ABB RAPID module: P781.mod

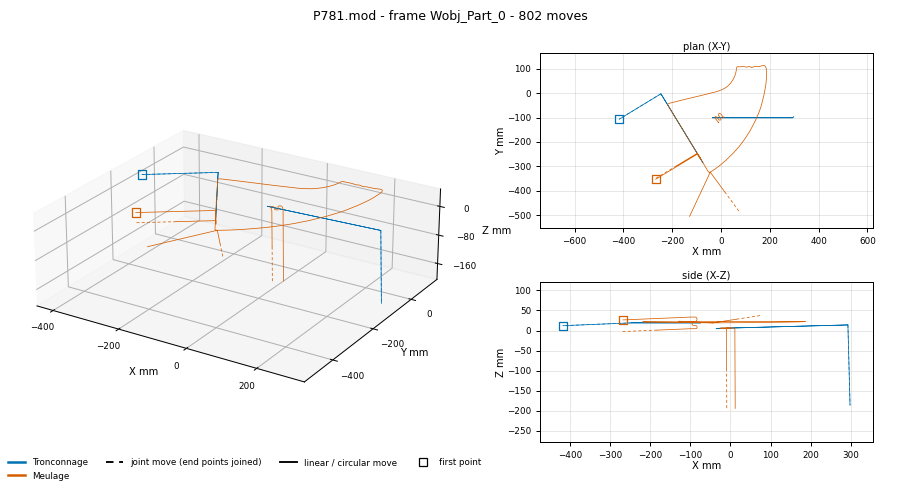
[picture p0: tool path of P781.mod in frame Wobj_Part_0, 802 of 822 moves have a stored position in this frame; points joined in program order, loops and branches not executed]
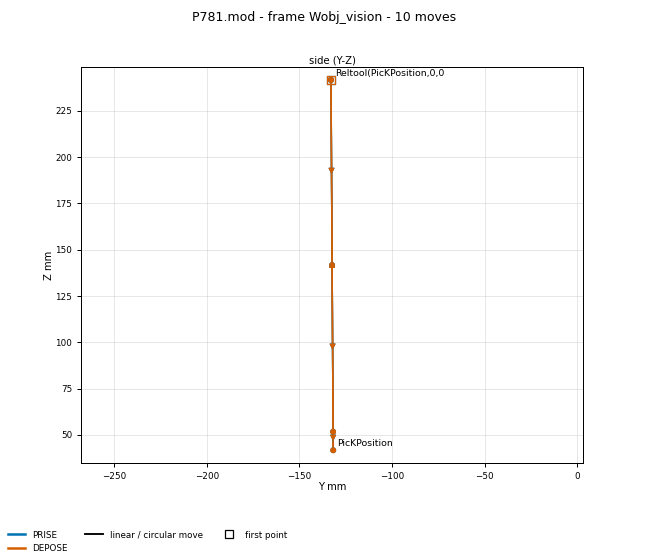
[picture p1: tool path of P781.mod in frame Wobj_vision, 10 of 822 moves have a stored position in this frame; points joined in program order, loops and branches not executed]
MODULE P781

    ! Nom         :P781
    ! Description :
    ! Créé le     :25/05/2023 15:38:47

    LOCAL CONST SPEEDDATA VitesseLente :=[10,500,0,0];
	LOCAL CONST SPEEDDATA VitesseRapide :=[30,500,0,0];
    !
    !Point de prise
    LOCAL PERS Robtarget PicKPosition := [[-23.1582873493958,-131.784324695273,41.7270241668186],[0.00267552588877119,-0.96306839839963,0.269238876085942,0.00159033618135217],[0,0,0,0],[8.999999E+09,8.999999E+09,8.999999E+09,8.999999E+09,8.999999E+09,8.999999E+09]];
	LOCAL PERS Pose Ref := [[0,0,0],[1,0,0,0]];
    !
    !Declaration des points de meulage

    !Tr_meulage_motif_1 : Meulage d'un motif
    LOCAL CONST Robtarget Tr_meulage_motif_1_0 := [[-96.4877265625,-249.765390625,33.67604296875],[0.626544891741501,-0.60457807117296,0.341537876614403,-0.353947359542544],[0,0,0,0],[8.999999E+09,8.999999E+09,8.999999E+09,8.999999E+09,8.999999E+09,8.999999E+09]];
    LOCAL CONST Robtarget Tr_meulage_motif_1_1 := [[-95.966875,-250.619046875,33.676046875],[0.626544891741501,-0.60457807117296,0.341537876614403,-0.353947359542544],[0,0,0,0],[8.999999E+09,8.999999E+09,8.999999E+09,8.999999E+09,8.999999E+09,8.999999E+09]];
    LOCAL CONST Robtarget Tr_meulage_motif_1_2 := [[-95.44603125,-251.4726875,33.6760546875],[0.626544891741501,-0.60457807117296,0.341537876614403,-0.353947359542544],[0,0,0,0],[8.999999E+09,8.999999E+09,8.999999E+09,8.999999E+09,8.999999E+09,8.999999E+09]];
    LOCAL CONST Robtarget Tr_meulage_motif_1_3 := [[-94.9251875,-252.32634375,33.6760625],[0.626544891741501,-0.60457807117296,0.341537876614403,-0.353947359542544],[0,0,0,0],[8.999999E+09,8.999999E+09,8.999999E+09,8.999999E+09,8.999999E+09,8.999999E+09]];
    LOCAL CONST Robtarget Tr_meulage_motif_1_4 := [[-94.40434375,-253.18,33.67606640625],[0.626544891741501,-0.60457807117296,0.341537876614403,-0.353947359542544],[0,0,0,0],[8.999999E+09,8.999999E+09,8.999999E+09,8.999999E+09,8.999999E+09,8.999999E+09]];
    LOCAL CONST Robtarget Tr_meulage_motif_1_5 := [[-93.8834921875,-254.033640625,33.67607421875],[0.626544891741501,-0.60457807117296,0.341537876614403,-0.353947359542544],[0,0,0,0],[8.999999E+09,8.999999E+09,8.999999E+09,8.999999E+09,8.999999E+09,8.999999E+09]];
    LOCAL CONST Robtarget Tr_meulage_motif_1_6 := [[-93.3626484375,-254.887296875,33.676078125],[0.626544891741501,-0.60457807117296,0.341537876614403,-0.353947359542544],[0,0,0,0],[8.999999E+09,8.999999E+09,8.999999E+09,8.999999E+09,8.999999E+09,8.999999E+09]];
    LOCAL CONST Robtarget Tr_meulage_motif_1_7 := [[-92.8418046875,-255.740953125,33.6760859375],[0.626544891741501,-0.60457807117296,0.341537876614403,-0.353947359542544],[0,0,0,0],[8.999999E+09,8.999999E+09,8.999999E+09,8.999999E+09,8.999999E+09,8.999999E+09]];
    LOCAL CONST Robtarget Tr_meulage_motif_1_8 := [[-92.320953125,-256.59459375,33.67608984375],[0.626544891741501,-0.60457807117296,0.341537876614403,-0.353947359542544],[0,0,0,0],[8.999999E+09,8.999999E+09,8.999999E+09,8.999999E+09,8.999999E+09,8.999999E+09]];
    LOCAL CONST Robtarget Tr_meulage_motif_1_9 := [[-91.800109375,-257.44825,33.67609765625],[0.626544891741501,-0.60457807117296,0.341537876614403,-0.353947359542544],[0,0,0,0],[8.999999E+09,8.999999E+09,8.999999E+09,8.999999E+09,8.999999E+09,8.999999E+09]];
    LOCAL CONST Robtarget Tr_meulage_motif_1_10 := [[-91.279265625,-258.30190625,33.6761015625],[0.626544891741501,-0.60457807117296,0.341537876614403,-0.353947359542544],[0,0,0,0],[8.999999E+09,8.999999E+09,8.999999E+09,8.999999E+09,8.999999E+09,8.999999E+09]];
    LOCAL CONST Robtarget Tr_meulage_motif_1_11 := [[-90.758421875,-259.155546875,33.676109375],[0.626544891741501,-0.60457807117296,0.341537876614403,-0.353947359542544],[0,0,0,0],[8.999999E+09,8.999999E+09,8.999999E+09,8.999999E+09,8.999999E+09,8.999999E+09]];
    LOCAL CONST Robtarget Tr_meulage_motif_1_12 := [[-90.2375703125,-260.009203125,33.67611328125],[0.626544891741501,-0.60457807117296,0.341537876614403,-0.353947359542544],[0,0,0,0],[8.999999E+09,8.999999E+09,8.999999E+09,8.999999E+09,8.999999E+09,8.999999E+09]];
    LOCAL CONST Robtarget Tr_meulage_motif_1_13 := [[-89.7167265625,-260.86284375,33.67612109375],[0.626544891741501,-0.60457807117296,0.341537876614403,-0.353947359542544],[0,0,0,0],[8.999999E+09,8.999999E+09,8.999999E+09,8.999999E+09,8.999999E+09,8.999999E+09]];
    LOCAL CONST Robtarget Tr_meulage_motif_1_14 := [[-89.1958828125,-261.7165,33.676125],[0.626544891741501,-0.60457807117296,0.341537876614403,-0.353947359542544],[0,0,0,0],[8.999999E+09,8.999999E+09,8.999999E+09,8.999999E+09,8.999999E+09,8.999999E+09]];
    LOCAL CONST Robtarget Tr_meulage_motif_1_15 := [[-88.67503125,-262.57015625,33.6761328125],[0.626544891741501,-0.60457807117296,0.341537876614403,-0.353947359542544],[0,0,0,0],[8.999999E+09,8.999999E+09,8.999999E+09,8.999999E+09,8.999999E+09,8.999999E+09]];
    LOCAL CONST Robtarget Tr_meulage_motif_1_16 := [[-88.1541875,-263.4238125,33.67613671875],[0.626544891741501,-0.60457807117296,0.341537876614403,-0.353947359542544],[0,0,0,0],[8.999999E+09,8.999999E+09,8.999999E+09,8.999999E+09,8.999999E+09,8.999999E+09]];
    LOCAL CONST Robtarget Tr_meulage_motif_1_17 := [[-87.63334375,-264.27746875,33.67614453125],[0.626544891741501,-0.60457807117296,0.341537876614403,-0.353947359542544],[0,0,0,0],[8.999999E+09,8.999999E+09,8.999999E+09,8.999999E+09,8.999999E+09,8.999999E+09]];
    LOCAL CONST Robtarget Tr_meulage_motif_1_18 := [[-87.1125,-265.13109375,33.6761484375],[0.626544891741501,-0.60457807117296,0.341537876614403,-0.353947359542544],[0,0,0,0],[8.999999E+09,8.999999E+09,8.999999E+09,8.999999E+09,8.999999E+09,8.999999E+09]];
    LOCAL CONST Robtarget Tr_meulage_motif_1_19 := [[-86.59221875,-265.976375,33.56562890625],[0.626544891741501,-0.60457807117296,0.341537876614403,-0.353947359542544],[0,0,0,0],[8.999999E+09,8.999999E+09,8.999999E+09,8.999999E+09,8.999999E+09,8.999999E+09]];
    LOCAL CONST Robtarget Tr_meulage_motif_1_20 := [[-86.0929296875,-266.78053125,33.35457421875],[0.626544891741501,-0.60457807117296,0.341537876614403,-0.353947359542544],[0,0,0,0],[8.999999E+09,8.999999E+09,8.999999E+09,8.999999E+09,8.999999E+09,8.999999E+09]];
    LOCAL CONST Robtarget Tr_meulage_motif_1_21 := [[-85.640671875,-267.5035,33.08290234375],[0.626544891741501,-0.60457807117296,0.341537876614403,-0.353947359542544],[0,0,0,0],[8.999999E+09,8.999999E+09,8.999999E+09,8.999999E+09,8.999999E+09,8.999999E+09]];
    LOCAL CONST Robtarget Tr_meulage_motif_1_22 := [[-85.241828125,-268.13865625,32.807140625],[0.626544891741501,-0.60457807117296,0.341537876614403,-0.353947359542544],[0,0,0,0],[8.999999E+09,8.999999E+09,8.999999E+09,8.999999E+09,8.999999E+09,8.999999E+09]];
    LOCAL CONST Robtarget Tr_meulage_motif_1_23 := [[-84.6499296875,-269.06734375,32.1913984375],[0.626544891741501,-0.60457807117296,0.341537876614403,-0.353947359542544],[0,0,0,0],[8.999999E+09,8.999999E+09,8.999999E+09,8.999999E+09,8.999999E+09,8.999999E+09]];
    LOCAL CONST Robtarget Tr_meulage_motif_1_24 := [[-84.091328125,-269.9259375,31.344267578125],[0.626544891741501,-0.60457807117296,0.341537876614403,-0.353947359542544],[0,0,0,0],[8.999999E+09,8.999999E+09,8.999999E+09,8.999999E+09,8.999999E+09,8.999999E+09]];
    LOCAL CONST Robtarget Tr_meulage_motif_1_25 := [[-83.619234375,-270.630875,30.321025390625],[0.626544891741501,-0.60457807117296,0.341537876614403,-0.353947359542544],[0,0,0,0],[8.999999E+09,8.999999E+09,8.999999E+09,8.999999E+09,8.999999E+09,8.999999E+09]];
    LOCAL CONST Robtarget Tr_meulage_motif_1_26 := [[-83.3316328125,-271.02725,29.2055234375],[0.626544891741501,-0.60457807117296,0.341537876614403,-0.353947359542544],[0,0,0,0],[8.999999E+09,8.999999E+09,8.999999E+09,8.999999E+09,8.999999E+09,8.999999E+09]];
    LOCAL CONST Robtarget Tr_meulage_motif_1_27 := [[-83.2967421875,-271.03765625,28.509982421875],[0.626544891741501,-0.60457807117296,0.341537876614403,-0.353947359542544],[0,0,0,0],[8.999999E+09,8.999999E+09,8.999999E+09,8.999999E+09,8.999999E+09,8.999999E+09]];
    LOCAL CONST Robtarget Tr_meulage_motif_1_28 := [[-83.276984375,-271.025625,27.84913671875],[0.626544891741501,-0.60457807117296,0.341537876614403,-0.353947359542544],[0,0,0,0],[8.999999E+09,8.999999E+09,8.999999E+09,8.999999E+09,8.999999E+09,8.999999E+09]];
    LOCAL CONST Robtarget Tr_meulage_motif_1_29 := [[-83.2858125,-270.96671875,27.188447265625],[0.626544891741501,-0.60457807117296,0.341537876614403,-0.353947359542544],[0,0,0,0],[8.999999E+09,8.999999E+09,8.999999E+09,8.999999E+09,8.999999E+09,8.999999E+09]];
    LOCAL CONST Robtarget Tr_meulage_motif_1_30 := [[-83.512390625,-270.52134375,26.087369140625],[0.626544891741501,-0.60457807117296,0.341537876614403,-0.353947359542544],[0,0,0,0],[8.999999E+09,8.999999E+09,8.999999E+09,8.999999E+09,8.999999E+09,8.999999E+09]];
    LOCAL CONST Robtarget Tr_meulage_motif_1_31 := [[-83.928484375,-269.77175,25.081357421875],[0.626544891741501,-0.60457807117296,0.341537876614403,-0.353947359542544],[0,0,0,0],[8.999999E+09,8.999999E+09,8.999999E+09,8.999999E+09,8.999999E+09,8.999999E+09]];
    LOCAL CONST Robtarget Tr_meulage_motif_1_32 := [[-84.4367578125,-268.883,24.252982421875],[0.626544891741501,-0.60457807117296,0.341537876614403,-0.353947359542544],[0,0,0,0],[8.999999E+09,8.999999E+09,8.999999E+09,8.999999E+09,8.999999E+09,8.999999E+09]];
    LOCAL CONST Robtarget Tr_meulage_motif_1_33 := [[-84.782796875,-268.28925,23.857470703125],[0.626544891741501,-0.60457807117296,0.341537876614403,-0.353947359542544],[0,0,0,0],[8.999999E+09,8.999999E+09,8.999999E+09,8.999999E+09,8.999999E+09,8.999999E+09]];
    LOCAL CONST Robtarget Tr_meulage_motif_1_34 := [[-85.371453125,-267.29171875,23.370232421875],[0.626544891741501,-0.60457807117296,0.341537876614403,-0.353947359542544],[0,0,0,0],[8.999999E+09,8.999999E+09,8.999999E+09,8.999999E+09,8.999999E+09,8.999999E+09]];
    LOCAL CONST Robtarget Tr_meulage_motif_1_35 := [[-85.8036953125,-266.56553125,23.106294921875],[0.626544891741501,-0.60457807117296,0.341537876614403,-0.353947359542544],[0,0,0,0],[8.999999E+09,8.999999E+09,8.999999E+09,8.999999E+09,8.999999E+09,8.999999E+09]];
    LOCAL CONST Robtarget Tr_meulage_motif_1_36 := [[-86.283015625,-265.76621875,22.9019453125],[0.626544891741501,-0.60457807117296,0.341537876614403,-0.353947359542544],[0,0,0,0],[8.999999E+09,8.999999E+09,8.999999E+09,8.999999E+09,8.999999E+09,8.999999E+09]];
    LOCAL CONST Robtarget Tr_meulage_motif_1_37 := [[-86.791015625,-264.9263125,22.7934140625],[0.626544891741501,-0.60457807117296,0.341537876614403,-0.353947359542544],[0,0,0,0],[8.999999E+09,8.999999E+09,8.999999E+09,8.999999E+09,8.999999E+09,8.999999E+09]];
    LOCAL CONST Robtarget Tr_meulage_motif_1_38 := [[-87.3046796875,-264.077,22.682880859375],[0.626544891741501,-0.60457807117296,0.341537876614403,-0.353947359542544],[0,0,0,0],[8.999999E+09,8.999999E+09,8.999999E+09,8.999999E+09,8.999999E+09,8.999999E+09]];
    LOCAL CONST Robtarget Tr_meulage_motif_1_39 := [[-87.8255234375,-263.22334375,22.682875],[0.626544891741501,-0.60457807117296,0.341537876614403,-0.353947359542544],[0,0,0,0],[8.999999E+09,8.999999E+09,8.999999E+09,8.999999E+09,8.999999E+09,8.999999E+09]];
    LOCAL CONST Robtarget Tr_meulage_motif_1_40 := [[-88.346375,-262.3696875,22.682869140625],[0.626544891741501,-0.60457807117296,0.341537876614403,-0.353947359542544],[0,0,0,0],[8.999999E+09,8.999999E+09,8.999999E+09,8.999999E+09,8.999999E+09,8.999999E+09]];
    LOCAL CONST Robtarget Tr_meulage_motif_1_41 := [[-88.86721875,-261.516046875,22.68286328125],[0.626544891741501,-0.60457807117296,0.341537876614403,-0.353947359542544],[0,0,0,0],[8.999999E+09,8.999999E+09,8.999999E+09,8.999999E+09,8.999999E+09,8.999999E+09]];
    LOCAL CONST Robtarget Tr_meulage_motif_1_42 := [[-89.3880625,-260.662390625,22.682857421875],[0.626544891741501,-0.60457807117296,0.341537876614403,-0.353947359542544],[0,0,0,0],[8.999999E+09,8.999999E+09,8.999999E+09,8.999999E+09,8.999999E+09,8.999999E+09]];
    LOCAL CONST Robtarget Tr_meulage_motif_1_43 := [[-89.9089140625,-259.80875,22.6828515625],[0.626544891741501,-0.60457807117296,0.341537876614403,-0.353947359542544],[0,0,0,0],[8.999999E+09,8.999999E+09,8.999999E+09,8.999999E+09,8.999999E+09,8.999999E+09]];
    LOCAL CONST Robtarget Tr_meulage_motif_1_44 := [[-90.4297578125,-258.95509375,22.682845703125],[0.626544891741501,-0.60457807117296,0.341537876614403,-0.353947359542544],[0,0,0,0],[8.999999E+09,8.999999E+09,8.999999E+09,8.999999E+09,8.999999E+09,8.999999E+09]];
    LOCAL CONST Robtarget Tr_meulage_motif_1_45 := [[-90.9506015625,-258.1014375,22.68283984375],[0.626544891741501,-0.60457807117296,0.341537876614403,-0.353947359542544],[0,0,0,0],[8.999999E+09,8.999999E+09,8.999999E+09,8.999999E+09,8.999999E+09,8.999999E+09]];
    LOCAL CONST Robtarget Tr_meulage_motif_1_46 := [[-91.4714453125,-257.247796875,22.682833984375],[0.626544891741501,-0.60457807117296,0.341537876614403,-0.353947359542544],[0,0,0,0],[8.999999E+09,8.999999E+09,8.999999E+09,8.999999E+09,8.999999E+09,8.999999E+09]];
    LOCAL CONST Robtarget Tr_meulage_motif_1_47 := [[-91.992296875,-256.394140625,22.682828125],[0.626544891741501,-0.60457807117296,0.341537876614403,-0.353947359542544],[0,0,0,0],[8.999999E+09,8.999999E+09,8.999999E+09,8.999999E+09,8.999999E+09,8.999999E+09]];
    LOCAL CONST Robtarget Tr_meulage_motif_1_48 := [[-92.513140625,-255.5405,22.682822265625],[0.626544891741501,-0.60457807117296,0.341537876614403,-0.353947359542544],[0,0,0,0],[8.999999E+09,8.999999E+09,8.999999E+09,8.999999E+09,8.999999E+09,8.999999E+09]];
    LOCAL CONST Robtarget Tr_meulage_motif_1_49 := [[-93.0268046875,-254.691171875,22.572291015625],[0.626544891741501,-0.60457807117296,0.341537876614403,-0.353947359542544],[0,0,0,0],[8.999999E+09,8.999999E+09,8.999999E+09,8.999999E+09,8.999999E+09,8.999999E+09]];
    LOCAL CONST Robtarget Tr_meulage_motif_1_50 := [[-93.5134765625,-253.87934375,22.3612265625],[0.626544891741501,-0.60457807117296,0.341537876614403,-0.353947359542544],[0,0,0,0],[8.999999E+09,8.999999E+09,8.999999E+09,8.999999E+09,8.999999E+09,8.999999E+09]];
    LOCAL CONST Robtarget Tr_meulage_motif_1_51 := [[-93.9494921875,-253.14646875,22.089544921875],[0.626544891741501,-0.60457807117296,0.341537876614403,-0.353947359542544],[0,0,0,0],[8.999999E+09,8.999999E+09,8.999999E+09,8.999999E+09,8.999999E+09,8.999999E+09]];
    LOCAL CONST Robtarget Tr_meulage_motif_1_52 := [[-94.310984375,-252.533546875,21.7855703125],[0.626544891741501,-0.60457807117296,0.341537876614403,-0.353947359542544],[0,0,0,0],[8.999999E+09,8.999999E+09,8.999999E+09,8.999999E+09,8.999999E+09,8.999999E+09]];
    LOCAL CONST Robtarget Tr_meulage_motif_1_53 := [[-94.8299921875,-251.63840625,21.123439453125],[0.626544891741501,-0.60457807117296,0.341537876614403,-0.353947359542544],[0,0,0,0],[8.999999E+09,8.999999E+09,8.999999E+09,8.999999E+09,8.999999E+09,8.999999E+09]];
    LOCAL CONST Robtarget Tr_meulage_motif_1_54 := [[-95.2728125,-250.85203125,20.222048828125],[0.626544891741501,-0.60457807117296,0.341537876614403,-0.353947359542544],[0,0,0,0],[8.999999E+09,8.999999E+09,8.999999E+09,8.999999E+09,8.999999E+09,8.999999E+09]];
    LOCAL CONST Robtarget Tr_meulage_motif_1_55 := [[-95.5201953125,-250.376296875,19.176654296875],[0.626544891741501,-0.60457807117296,0.341537876614403,-0.353947359542544],[0,0,0,0],[8.999999E+09,8.999999E+09,8.999999E+09,8.999999E+09,8.999999E+09,8.999999E+09]];
    LOCAL CONST Robtarget Tr_meulage_motif_1_56 := [[-95.5957265625,-250.205921875,18.483859375],[0.626544891741501,-0.60457807117296,0.341537876614403,-0.353947359542544],[0,0,0,0],[8.999999E+09,8.999999E+09,8.999999E+09,8.999999E+09,8.999999E+09,8.999999E+09]];
    LOCAL CONST Robtarget Tr_meulage_motif_1_57 := [[-95.60596875,-250.137390625,17.71433203125],[0.626544891741501,-0.60457807117296,0.341537876614403,-0.353947359542544],[0,0,0,0],[8.999999E+09,8.999999E+09,8.999999E+09,8.999999E+09,8.999999E+09,8.999999E+09]];
    LOCAL CONST Robtarget Tr_meulage_motif_1_58 := [[-95.5481015625,-250.1805,16.944927734375],[0.626544891741501,-0.60457807117296,0.341537876614403,-0.353947359542544],[0,0,0,0],[8.999999E+09,8.999999E+09,8.999999E+09,8.999999E+09,8.999999E+09,8.999999E+09]];
    LOCAL CONST Robtarget Tr_meulage_motif_1_59 := [[-95.2964453125,-250.518484375,15.837359375],[0.626544891741501,-0.60457807117296,0.341537876614403,-0.353947359542544],[0,0,0,0],[8.999999E+09,8.999999E+09,8.999999E+09,8.999999E+09,8.999999E+09,8.999999E+09]];
    LOCAL CONST Robtarget Tr_meulage_motif_1_60 := [[-95.06315625,-250.8615,15.252033203125],[0.626544891741501,-0.60457807117296,0.341537876614403,-0.353947359542544],[0,0,0,0],[8.999999E+09,8.999999E+09,8.999999E+09,8.999999E+09,8.999999E+09,8.999999E+09]];
    LOCAL CONST Robtarget Tr_meulage_motif_1_61 := [[-94.57459375,-251.602625,14.36545703125],[0.626544891741501,-0.60457807117296,0.341537876614403,-0.353947359542544],[0,0,0,0],[8.999999E+09,8.999999E+09,8.999999E+09,8.999999E+09,8.999999E+09,8.999999E+09]];
    LOCAL CONST Robtarget Tr_meulage_motif_1_62 := [[-94.2571640625,-252.095046875,13.95140234375],[0.626544891741501,-0.60457807117296,0.341537876614403,-0.353947359542544],[0,0,0,0],[8.999999E+09,8.999999E+09,8.999999E+09,8.999999E+09,8.999999E+09,8.999999E+09]];
    LOCAL CONST Robtarget Tr_meulage_motif_1_63 := [[-93.6586484375,-253.0394375,13.4076484375],[0.626544891741501,-0.60457807117296,0.341537876614403,-0.353947359542544],[0,0,0,0],[8.999999E+09,8.999999E+09,8.999999E+09,8.999999E+09,8.999999E+09,8.999999E+09]];
    LOCAL CONST Robtarget Tr_meulage_motif_1_64 := [[-93.2198125,-253.7388125,13.112333984375],[0.626544891741501,-0.60457807117296,0.341537876614403,-0.353947359542544],[0,0,0,0],[8.999999E+09,8.999999E+09,8.999999E+09,8.999999E+09,8.999999E+09,8.999999E+09]];
    LOCAL CONST Robtarget Tr_meulage_motif_1_65 := [[-92.7282734375,-254.5306875,12.90799609375],[0.626544891741501,-0.60457807117296,0.341537876614403,-0.353947359542544],[0,0,0,0],[8.999999E+09,8.999999E+09,8.999999E+09,8.999999E+09,8.999999E+09,8.999999E+09]];
    LOCAL CONST Robtarget Tr_meulage_motif_1_66 := [[-92.2137890625,-255.366625,12.799474609375],[0.626544891741501,-0.60457807117296,0.341537876614403,-0.353947359542544],[0,0,0,0],[8.999999E+09,8.999999E+09,8.999999E+09,8.999999E+09,8.999999E+09,8.999999E+09]];
    LOCAL CONST Robtarget Tr_meulage_motif_1_67 := [[-91.6935078125,-256.21190625,12.6889541015625],[0.626544891741501,-0.60457807117296,0.341537876614403,-0.353947359542544],[0,0,0,0],[8.999999E+09,8.999999E+09,8.999999E+09,8.999999E+09,8.999999E+09,8.999999E+09]];
    LOCAL CONST Robtarget Tr_meulage_motif_1_68 := [[-91.1726640625,-257.0655625,12.6889599609375],[0.626544891741501,-0.60457807117296,0.341537876614403,-0.353947359542544],[0,0,0,0],[8.999999E+09,8.999999E+09,8.999999E+09,8.999999E+09,8.999999E+09,8.999999E+09]];
    LOCAL CONST Robtarget Tr_meulage_motif_1_69 := [[-90.6518203125,-257.91921875,12.6889658203125],[0.626544891741501,-0.60457807117296,0.341537876614403,-0.353947359542544],[0,0,0,0],[8.999999E+09,8.999999E+09,8.999999E+09,8.999999E+09,8.999999E+09,8.999999E+09]];
    LOCAL CONST Robtarget Tr_meulage_motif_1_70 := [[-90.1309765625,-258.772859375,12.6889716796875],[0.626544891741501,-0.60457807117296,0.341537876614403,-0.353947359542544],[0,0,0,0],[8.999999E+09,8.999999E+09,8.999999E+09,8.999999E+09,8.999999E+09,8.999999E+09]];
    LOCAL CONST Robtarget Tr_meulage_motif_1_71 := [[-89.610125,-259.626515625,12.6889775390625],[0.626544891741501,-0.60457807117296,0.341537876614403,-0.353947359542544],[0,0,0,0],[8.999999E+09,8.999999E+09,8.999999E+09,8.999999E+09,8.999999E+09,8.999999E+09]];
    LOCAL CONST Robtarget Tr_meulage_motif_1_72 := [[-89.08928125,-260.480171875,12.6889833984375],[0.626544891741501,-0.60457807117296,0.341537876614403,-0.353947359542544],[0,0,0,0],[8.999999E+09,8.999999E+09,8.999999E+09,8.999999E+09,8.999999E+09,8.999999E+09]];
    LOCAL CONST Robtarget Tr_meulage_motif_1_73 := [[-88.5684375,-261.3338125,12.6889892578125],[0.626544891741501,-0.60457807117296,0.341537876614403,-0.353947359542544],[0,0,0,0],[8.999999E+09,8.999999E+09,8.999999E+09,8.999999E+09,8.999999E+09,8.999999E+09]];
    LOCAL CONST Robtarget Tr_meulage_motif_1_74 := [[-88.0475859375,-262.18746875,12.6889951171875],[0.626544891741501,-0.60457807117296,0.341537876614403,-0.353947359542544],[0,0,0,0],[8.999999E+09,8.999999E+09,8.999999E+09,8.999999E+09,8.999999E+09,8.999999E+09]];
    LOCAL CONST Robtarget Tr_meulage_motif_1_75 := [[-87.5267421875,-263.041125,12.6890009765625],[0.626544891741501,-0.60457807117296,0.341537876614403,-0.353947359542544],[0,0,0,0],[8.999999E+09,8.999999E+09,8.999999E+09,8.999999E+09,8.999999E+09,8.999999E+09]];
    LOCAL CONST Robtarget Tr_meulage_motif_1_76 := [[-87.0058984375,-263.89478125,12.6890068359375],[0.626544891741501,-0.60457807117296,0.341537876614403,-0.353947359542544],[0,0,0,0],[8.999999E+09,8.999999E+09,8.999999E+09,8.999999E+09,8.999999E+09,8.999999E+09]];
    LOCAL CONST Robtarget Tr_meulage_motif_1_77 := [[-86.4850546875,-264.74840625,12.6890126953125],[0.626544891741501,-0.60457807117296,0.341537876614403,-0.353947359542544],[0,0,0,0],[8.999999E+09,8.999999E+09,8.999999E+09,8.999999E+09,8.999999E+09,8.999999E+09]];
    LOCAL CONST Robtarget Tr_meulage_motif_1_78 := [[-85.9647734375,-265.59371875,12.5784931640625],[0.626544891741501,-0.60457807117296,0.341537876614403,-0.353947359542544],[0,0,0,0],[8.999999E+09,8.999999E+09,8.999999E+09,8.999999E+09,8.999999E+09,8.999999E+09]];
    LOCAL CONST Robtarget Tr_meulage_motif_1_79 := [[-85.465484375,-266.39784375,12.3674404296875],[0.626544891741501,-0.60457807117296,0.341537876614403,-0.353947359542544],[0,0,0,0],[8.999999E+09,8.999999E+09,8.999999E+09,8.999999E+09,8.999999E+09,8.999999E+09]];
    LOCAL CONST Robtarget Tr_meulage_motif_1_80 := [[-85.0132265625,-267.1208125,12.0957685546875],[0.626544891741501,-0.60457807117296,0.341537876614403,-0.353947359542544],[0,0,0,0],[8.999999E+09,8.999999E+09,8.999999E+09,8.999999E+09,8.999999E+09,8.999999E+09]];
    LOCAL CONST Robtarget Tr_meulage_motif_1_81 := [[-84.6143828125,-267.75596875,11.82000390625],[0.626544891741501,-0.60457807117296,0.341537876614403,-0.353947359542544],[0,0,0,0],[8.999999E+09,8.999999E+09,8.999999E+09,8.999999E+09,8.999999E+09,8.999999E+09]];
    LOCAL CONST Robtarget Tr_meulage_motif_1_82 := [[-84.022484375,-268.68465625,11.2042626953125],[0.626544891741501,-0.60457807117296,0.341537876614403,-0.353947359542544],[0,0,0,0],[8.999999E+09,8.999999E+09,8.999999E+09,8.999999E+09,8.999999E+09,8.999999E+09]];
    LOCAL CONST Robtarget Tr_meulage_motif_1_83 := [[-83.4974765625,-269.4850625,10.31084765625],[0.626544891741501,-0.60457807117296,0.341537876614403,-0.353947359542544],[0,0,0,0],[8.999999E+09,8.999999E+09,8.999999E+09,8.999999E+09,8.999999E+09,8.999999E+09]];
    LOCAL CONST Robtarget Tr_meulage_motif_1_84 := [[-83.147765625,-269.98525,9.2255166015625],[0.626544891741501,-0.60457807117296,0.341537876614403,-0.353947359542544],[0,0,0,0],[8.999999E+09,8.999999E+09,8.999999E+09,8.999999E+09,8.999999E+09,8.999999E+09]];
    LOCAL CONST Robtarget Tr_meulage_motif_1_85 := [[-83.030171875,-270.11184375,8.2417451171875],[0.626544891741501,-0.60457807117296,0.341537876614403,-0.353947359542544],[0,0,0,0],[8.999999E+09,8.999999E+09,8.999999E+09,8.999999E+09,8.999999E+09,8.999999E+09]];
    LOCAL CONST Robtarget Tr_meulage_motif_1_86 := [[-83.09253125,-269.99590625,8.0372138671875],[0.626544891741501,-0.60457807117296,0.341537876614403,-0.353947359542544],[0,0,0,0],[8.999999E+09,8.999999E+09,8.999999E+09,8.999999E+09,8.999999E+09,8.999999E+09]];
    LOCAL CONST Robtarget Tr_meulage_motif_1_87 := [[-83.1350859375,-269.87734375,7.311251953125],[0.626544891741501,-0.60457807117296,0.341537876614403,-0.353947359542544],[0,0,0,0],[8.999999E+09,8.999999E+09,8.999999E+09,8.999999E+09,8.999999E+09,8.999999E+09]];
    LOCAL CONST Robtarget Tr_meulage_motif_1_88 := [[-83.4633515625,-269.276375,6.37491552734375],[0.626544891741501,-0.60457807117296,0.341537876614403,-0.353947359542544],[0,0,0,0],[8.999999E+09,8.999999E+09,8.999999E+09,8.999999E+09,8.999999E+09,8.999999E+09]];
    LOCAL CONST Robtarget Tr_meulage_motif_1_89 := [[-83.7399296875,-268.79190625,5.9113837890625],[0.626544891741501,-0.60457807117296,0.341537876614403,-0.353947359542544],[0,0,0,0],[8.999999E+09,8.999999E+09,8.999999E+09,8.999999E+09,8.999999E+09,8.999999E+09]];
    LOCAL CONST Robtarget Tr_meulage_motif_1_90 := [[-84.312796875,-267.81734375,5.3812646484375],[0.626544891741501,-0.60457807117296,0.341537876614403,-0.353947359542544],[0,0,0,0],[8.999999E+09,8.999999E+09,8.999999E+09,8.999999E+09,8.999999E+09,8.999999E+09]];
    LOCAL CONST Robtarget Tr_meulage_motif_1_91 := [[-84.7450390625,-267.09115625,5.11732763671875],[0.626544891741501,-0.60457807117296,0.341537876614403,-0.353947359542544],[0,0,0,0],[8.999999E+09,8.999999E+09,8.999999E+09,8.999999E+09,8.999999E+09,8.999999E+09]];
    LOCAL CONST Robtarget Tr_meulage_motif_1_92 := [[-85.224359375,-266.29184375,4.912978515625],[0.626544891741501,-0.60457807117296,0.341537876614403,-0.353947359542544],[0,0,0,0],[8.999999E+09,8.999999E+09,8.999999E+09,8.999999E+09,8.999999E+09,8.999999E+09]];
    LOCAL CONST Robtarget Tr_meulage_motif_1_93 := [[-85.732359375,-265.4519375,4.80444580078125],[0.626544891741501,-0.60457807117296,0.341537876614403,-0.353947359542544],[0,0,0,0],[8.999999E+09,8.999999E+09,8.999999E+09,8.999999E+09,8.999999E+09,8.999999E+09]];
    LOCAL CONST Robtarget Tr_meulage_motif_1_94 := [[-86.2460234375,-264.602625,4.6939140625],[0.626544891741501,-0.60457807117296,0.341537876614403,-0.353947359542544],[0,0,0,0],[8.999999E+09,8.999999E+09,8.999999E+09,8.999999E+09,8.999999E+09,8.999999E+09]];
    LOCAL CONST Robtarget Tr_meulage_motif_1_95 := [[-86.7668671875,-263.749,4.69390771484375],[0.626544891741501,-0.60457807117296,0.341537876614403,-0.353947359542544],[0,0,0,0],[8.999999E+09,8.999999E+09,8.999999E+09,8.999999E+09,8.999999E+09,8.999999E+09]];
    LOCAL CONST Robtarget Tr_meulage_motif_1_96 := [[-87.28771875,-262.89534375,4.69390185546875],[0.626544891741501,-0.60457807117296,0.341537876614403,-0.353947359542544],[0,0,0,0],[8.999999E+09,8.999999E+09,8.999999E+09,8.999999E+09,8.999999E+09,8.999999E+09]];
    LOCAL CONST Robtarget Tr_meulage_motif_1_97 := [[-87.8085625,-262.0416875,4.69389599609375],[0.626544891741501,-0.60457807117296,0.341537876614403,-0.353947359542544],[0,0,0,0],[8.999999E+09,8.999999E+09,8.999999E+09,8.999999E+09,8.999999E+09,8.999999E+09]];
    LOCAL CONST Robtarget Tr_meulage_motif_1_98 := [[-88.32940625,-261.18803125,4.69389013671875],[0.626544891741501,-0.60457807117296,0.341537876614403,-0.353947359542544],[0,0,0,0],[8.999999E+09,8.999999E+09,8.999999E+09,8.999999E+09,8.999999E+09,8.999999E+09]];
    LOCAL CONST Robtarget Tr_meulage_motif_1_99 := [[-88.8502578125,-260.334375,4.69388427734375],[0.626544891741501,-0.60457807117296,0.341537876614403,-0.353947359542544],[0,0,0,0],[8.999999E+09,8.999999E+09,8.999999E+09,8.999999E+09,8.999999E+09,8.999999E+09]];
    LOCAL CONST Robtarget Tr_meulage_motif_1_100 := [[-89.3711015625,-259.480734375,4.69387841796875],[0.626544891741501,-0.60457807117296,0.341537876614403,-0.353947359542544],[0,0,0,0],[8.999999E+09,8.999999E+09,8.999999E+09,8.999999E+09,8.999999E+09,8.999999E+09]];
    LOCAL CONST Robtarget Tr_meulage_motif_1_101 := [[-89.8919453125,-258.627078125,4.69387255859375],[0.626544891741501,-0.60457807117296,0.341537876614403,-0.353947359542544],[0,0,0,0],[8.999999E+09,8.999999E+09,8.999999E+09,8.999999E+09,8.999999E+09,8.999999E+09]];
    LOCAL CONST Robtarget Tr_meulage_motif_1_102 := [[-90.4127890625,-257.7734375,4.69386669921875],[0.626544891741501,-0.60457807117296,0.341537876614403,-0.353947359542544],[0,0,0,0],[8.999999E+09,8.999999E+09,8.999999E+09,8.999999E+09,8.999999E+09,8.999999E+09]];
    LOCAL CONST Robtarget Tr_meulage_motif_1_103 := [[-90.933640625,-256.91978125,4.69386083984375],[0.626544891741501,-0.60457807117296,0.341537876614403,-0.353947359542544],[0,0,0,0],[8.999999E+09,8.999999E+09,8.999999E+09,8.999999E+09,8.999999E+09,8.999999E+09]];
    LOCAL CONST Robtarget Tr_meulage_motif_1_104 := [[-91.454484375,-256.066125,4.69385498046875],[0.626544891741501,-0.60457807117296,0.341537876614403,-0.353947359542544],[0,0,0,0],[8.999999E+09,8.999999E+09,8.999999E+09,8.999999E+09,8.999999E+09,8.999999E+09]];
    LOCAL CONST Robtarget Tr_meulage_motif_1_105 := [[-91.975328125,-255.212484375,4.69384912109375],[0.626544891741501,-0.60457807117296,0.341537876614403,-0.353947359542544],[0,0,0,0],[8.999999E+09,8.999999E+09,8.999999E+09,8.999999E+09,8.999999E+09,8.999999E+09]];
    LOCAL CONST Robtarget Tr_meulage_motif_1_106 := [[-92.4961796875,-254.358828125,4.69384326171875],[0.626544891741501,-0.60457807117296,0.341537876614403,-0.353947359542544],[0,0,0,0],[8.999999E+09,8.999999E+09,8.999999E+09,8.999999E+09,8.999999E+09,8.999999E+09]];
    LOCAL CONST Robtarget Tr_meulage_motif_1_107 := [[-93.0170234375,-253.505171875,4.69383740234375],[0.626544891741501,-0.60457807117296,0.341537876614403,-0.353947359542544],[0,0,0,0],[8.999999E+09,8.999999E+09,8.999999E+09,8.999999E+09,8.999999E+09,8.999999E+09]];
    LOCAL CONST Robtarget Tr_meulage_motif_1_108 := [[-93.5378671875,-252.65153125,4.69383154296875],[0.626544891741501,-0.60457807117296,0.341537876614403,-0.353947359542544],[0,0,0,0],[8.999999E+09,8.999999E+09,8.999999E+09,8.999999E+09,8.999999E+09,8.999999E+09]];
    LOCAL CONST Robtarget Tr_meulage_motif_1_109 := [[-94.0587109375,-251.797875,4.69382568359375],[0.626544891741501,-0.60457807117296,0.341537876614403,-0.353947359542544],[0,0,0,0],[8.999999E+09,8.999999E+09,8.999999E+09,8.999999E+09,8.999999E+09,8.999999E+09]];
    LOCAL CONST Robtarget Tr_meulage_motif_1_110 := [[-94.5795625,-250.94421875,4.69381982421875],[0.626544891741501,-0.60457807117296,0.341537876614403,-0.353947359542544],[0,0,0,0],[8.999999E+09,8.999999E+09,8.999999E+09,8.999999E+09,8.999999E+09,8.999999E+09]];
    LOCAL CONST Robtarget Tr_meulage_motif_1_111 := [[-95.10040625,-250.090578125,4.69381396484375],[0.626544891741501,-0.60457807117296,0.341537876614403,-0.353947359542544],[0,0,0,0],[8.999999E+09,8.999999E+09,8.999999E+09,8.999999E+09,8.999999E+09,8.999999E+09]];
    LOCAL CONST Robtarget Tr_meulage_motif_1_112 := [[-95.62125,-249.236921875,4.69380810546875],[0.626544891741501,-0.60457807117296,0.341537876614403,-0.353947359542544],[0,0,0,0],[8.999999E+09,8.999999E+09,8.999999E+09,8.999999E+09,8.999999E+09,8.999999E+09]];
    LOCAL CONST Robtarget Tr_meulage_motif_1_113 := [[-96.1421015625,-248.383265625,4.6938017578125],[0.626544891741501,-0.60457807117296,0.341537876614403,-0.353947359542544],[0,0,0,0],[8.999999E+09,8.999999E+09,8.999999E+09,8.999999E+09,8.999999E+09,8.999999E+09]];
    LOCAL CONST Robtarget Tr_meulage_motif_1_114 := [[-96.6629453125,-247.529625,4.6937958984375],[0.626544891741501,-0.60457807117296,0.341537876614403,-0.353947359542544],[0,0,0,0],[8.999999E+09,8.999999E+09,8.999999E+09,8.999999E+09,8.999999E+09,8.999999E+09]];
    LOCAL CONST Robtarget Tr_meulage_motif_1_115 := [[-97.1837890625,-246.67596875,4.6937900390625],[0.626544891741501,-0.60457807117296,0.341537876614403,-0.353947359542544],[0,0,0,0],[8.999999E+09,8.999999E+09,8.999999E+09,8.999999E+09,8.999999E+09,8.999999E+09]];

    !Tr_meulage_motif_2 : Meulage d'un motif
    LOCAL CONST Robtarget Tr_meulage_motif_2_0 := [[11.059822265625,-100.7916484375,6.14594775390625],[1.9380529697738E-05,0.00227567224534522,0.00851606674262758,-0.999961148018993],[0,0,0,0],[8.999999E+09,8.999999E+09,8.999999E+09,8.999999E+09,8.999999E+09,8.999999E+09]];
    LOCAL CONST Robtarget Tr_meulage_motif_2_1 := [[10.444326171875,-100.0036640625,6.16165283203125],[1.9380529697738E-05,0.00227567224534522,0.00851606674262758,-0.999961148018993],[0,0,0,0],[8.999999E+09,8.999999E+09,8.999999E+09,8.999999E+09,8.999999E+09,8.999999E+09]];
    LOCAL CONST Robtarget Tr_meulage_motif_2_2 := [[9.828830078125,-99.2156875,6.17735791015625],[1.9380529697738E-05,0.00227567224534522,0.00851606674262758,-0.999961148018993],[0,0,0,0],[8.999999E+09,8.999999E+09,8.999999E+09,8.999999E+09,8.999999E+09,8.999999E+09]];
    LOCAL CONST Robtarget Tr_meulage_motif_2_3 := [[9.2133349609375,-98.427703125,6.19306298828125],[1.9380529697738E-05,0.00227567224534522,0.00851606674262758,-0.999961148018993],[0,0,0,0],[8.999999E+09,8.999999E+09,8.999999E+09,8.999999E+09,8.999999E+09,8.999999E+09]];
    LOCAL CONST Robtarget Tr_meulage_motif_2_4 := [[8.5978388671875,-97.63971875,6.20876806640625],[1.9380529697738E-05,0.00227567224534522,0.00851606674262758,-0.999961148018993],[0,0,0,0],[8.999999E+09,8.999999E+09,8.999999E+09,8.999999E+09,8.999999E+09,8.999999E+09]];
    LOCAL CONST Robtarget Tr_meulage_motif_2_5 := [[7.9823427734375,-96.851734375,6.22447314453125],[1.9380529697738E-05,0.00227567224534522,0.00851606674262758,-0.999961148018993],[0,0,0,0],[8.999999E+09,8.999999E+09,8.999999E+09,8.999999E+09,8.999999E+09,8.999999E+09]];
    LOCAL CONST Robtarget Tr_meulage_motif_2_6 := [[7.3668466796875,-96.06375,6.24017822265625],[1.9380529697738E-05,0.00227567224534522,0.00851606674262758,-0.999961148018993],[0,0,0,0],[8.999999E+09,8.999999E+09,8.999999E+09,8.999999E+09,8.999999E+09,8.999999E+09]];
    LOCAL CONST Robtarget Tr_meulage_motif_2_7 := [[6.75135107421875,-95.275765625,6.2558828125],[1.9380529697738E-05,0.00227567224534522,0.00851606674262758,-0.999961148018993],[0,0,0,0],[8.999999E+09,8.999999E+09,8.999999E+09,8.999999E+09,8.999999E+09,8.999999E+09]];
    LOCAL CONST Robtarget Tr_meulage_motif_2_8 := [[6.13585498046875,-94.48778125,6.271587890625],[1.9380529697738E-05,0.00227567224534522,0.00851606674262758,-0.999961148018993],[0,0,0,0],[8.999999E+09,8.999999E+09,8.999999E+09,8.999999E+09,8.999999E+09,8.999999E+09]];
    LOCAL CONST Robtarget Tr_meulage_motif_2_9 := [[5.520359375,-93.699796875,6.28729296875],[1.9380529697738E-05,0.00227567224534522,0.00851606674262758,-0.999961148018993],[0,0,0,0],[8.999999E+09,8.999999E+09,8.999999E+09,8.999999E+09,8.999999E+09,8.999999E+09]];
    LOCAL CONST Robtarget Tr_meulage_motif_2_10 := [[4.90486328125,-92.9118125,6.302998046875],[1.9380529697738E-05,0.00227567224534522,0.00851606674262758,-0.999961148018993],[0,0,0,0],[8.999999E+09,8.999999E+09,8.999999E+09,8.999999E+09,8.999999E+09,8.999999E+09]];
    LOCAL CONST Robtarget Tr_meulage_motif_2_11 := [[4.28936767578125,-92.123828125,6.318703125],[1.9380529697738E-05,0.00227567224534522,0.00851606674262758,-0.999961148018993],[0,0,0,0],[8.999999E+09,8.999999E+09,8.999999E+09,8.999999E+09,8.999999E+09,8.999999E+09]];
    LOCAL CONST Robtarget Tr_meulage_motif_2_12 := [[3.67387158203125,-91.3358515625,6.334408203125],[1.9380529697738E-05,0.00227567224534522,0.00851606674262758,-0.999961148018993],[0,0,0,0],[8.999999E+09,8.999999E+09,8.999999E+09,8.999999E+09,8.999999E+09,8.999999E+09]];
    LOCAL CONST Robtarget Tr_meulage_motif_2_13 := [[3.05837573242187,-90.5478671875,6.35011279296875],[1.9380529697738E-05,0.00227567224534522,0.00851606674262758,-0.999961148018993],[0,0,0,0],[8.999999E+09,8.999999E+09,8.999999E+09,8.999999E+09,8.999999E+09,8.999999E+09]];
    LOCAL CONST Robtarget Tr_meulage_motif_2_14 := [[2.4428798828125,-89.7598828125,6.36581787109375],[1.9380529697738E-05,0.00227567224534522,0.00851606674262758,-0.999961148018993],[0,0,0,0],[8.999999E+09,8.999999E+09,8.999999E+09,8.999999E+09,8.999999E+09,8.999999E+09]];
    LOCAL CONST Robtarget Tr_meulage_motif_2_15 := [[1.82738403320313,-88.9718984375,6.38152294921875],[1.9380529697738E-05,0.00227567224534522,0.00851606674262758,-0.999961148018993],[0,0,0,0],[8.999999E+09,8.999999E+09,8.999999E+09,8.999999E+09,8.999999E+09,8.999999E+09]];
    LOCAL CONST Robtarget Tr_meulage_motif_2_16 := [[1.21188806152344,-88.1839140625,6.39722802734375],[1.9380529697738E-05,0.00227567224534522,0.00851606674262758,-0.999961148018993],[0,0,0,0],[8.999999E+09,8.999999E+09,8.999999E+09,8.999999E+09,8.999999E+09,8.999999E+09]];
    LOCAL CONST Robtarget Tr_meulage_motif_2_17 := [[0.596392211914063,-87.3959296875,6.41293310546875],[1.9380529697738E-05,0.00227567224534522,0.00851606674262758,-0.999961148018993],[0,0,0,0],[8.999999E+09,8.999999E+09,8.999999E+09,8.999999E+09,8.999999E+09,8.999999E+09]];
    LOCAL CONST Robtarget Tr_meulage_motif_2_18 := [[-0.0191036529541016,-86.6079453125,6.42863818359375],[1.9380529697738E-05,0.00227567224534522,0.00851606674262758,-0.999961148018993],[0,0,0,0],[8.999999E+09,8.999999E+09,8.999999E+09,8.999999E+09,8.999999E+09,8.999999E+09]];
    LOCAL CONST Robtarget Tr_meulage_motif_2_19 := [[-0.717185119628906,-85.893875,6.44274560546875],[1.9380529697738E-05,0.00227567224534522,0.00851606674262758,-0.999961148018993],[0,0,0,0],[8.999999E+09,8.999999E+09,8.999999E+09,8.999999E+09,8.999999E+09,8.999999E+09]];
    LOCAL CONST Robtarget Tr_meulage_motif_2_20 := [[-1.46619714355469,-85.2780078125,6.454783203125],[1.9380529697738E-05,0.00227567224534522,0.00851606674262758,-0.999961148018993],[0,0,0,0],[8.999999E+09,8.999999E+09,8.999999E+09,8.999999E+09,8.999999E+09,8.999999E+09]];
    LOCAL CONST Robtarget Tr_meulage_motif_2_21 := [[-2.20529296875,-84.773359375,6.4645361328125],[1.9380529697738E-05,0.00227567224534522,0.00851606674262758,-0.999961148018993],[0,0,0,0],[8.999999E+09,8.999999E+09,8.999999E+09,8.999999E+09,8.999999E+09,8.999999E+09]];
    LOCAL CONST Robtarget Tr_meulage_motif_2_22 := [[-2.884353515625,-84.35221875,6.47261962890625],[1.9380529697738E-05,0.00227567224534522,0.00851606674262758,-0.999961148018993],[0,0,0,0],[8.999999E+09,8.999999E+09,8.999999E+09,8.999999E+09,8.999999E+09,8.999999E+09]];
    LOCAL CONST Robtarget Tr_meulage_motif_2_23 := [[-4.0476455078125,-83.8637265625,6.48166357421875],[1.9380529697738E-05,0.00227567224534522,0.00851606674262758,-0.999961148018993],[0,0,0,0],[8.999999E+09,8.999999E+09,8.999999E+09,8.999999E+09,8.999999E+09,8.999999E+09]];
    LOCAL CONST Robtarget Tr_meulage_motif_2_24 := [[-5.34590771484375,-83.5785390625,6.4863955078125],[1.9380529697738E-05,0.00227567224534522,0.00851606674262758,-0.999961148018993],[0,0,0,0],[8.999999E+09,8.999999E+09,8.999999E+09,8.999999E+09,8.999999E+09,8.999999E+09]];
    LOCAL CONST Robtarget Tr_meulage_motif_2_25 := [[-6.67459326171875,-83.540640625,6.4860009765625],[1.9380529697738E-05,0.00227567224534522,0.00851606674262758,-0.999961148018993],[0,0,0,0],[8.999999E+09,8.999999E+09,8.999999E+09,8.999999E+09,8.999999E+09,8.999999E+09]];
    LOCAL CONST Robtarget Tr_meulage_motif_2_26 := [[-7.85476318359375,-83.842828125,6.478724609375],[1.9380529697738E-05,0.00227567224534522,0.00851606674262758,-0.999961148018993],[0,0,0,0],[8.999999E+09,8.999999E+09,8.999999E+09,8.999999E+09,8.999999E+09,8.999999E+09]];
    LOCAL CONST Robtarget Tr_meulage_motif_2_27 := [[-8.4199404296875,-84.2497734375,6.46983251953125],[1.9380529697738E-05,0.00227567224534522,0.00851606674262758,-0.999961148018993],[0,0,0,0],[8.999999E+09,8.999999E+09,8.999999E+09,8.999999E+09,8.999999E+09,8.999999E+09]];
    LOCAL CONST Robtarget Tr_meulage_motif_2_28 := [[-8.94109765625,-84.656671875,6.46097998046875],[1.9380529697738E-05,0.00227567224534522,0.00851606674262758,-0.999961148018993],[0,0,0,0],[8.999999E+09,8.999999E+09,8.999999E+09,8.999999E+09,8.999999E+09,8.999999E+09]];
    LOCAL CONST Robtarget Tr_meulage_motif_2_29 := [[-9.4283564453125,-85.10671875,6.45126806640625],[1.9380529697738E-05,0.00227567224534522,0.00851606674262758,-0.999961148018993],[0,0,0,0],[8.999999E+09,8.999999E+09,8.999999E+09,8.999999E+09,8.999999E+09,8.999999E+09]];
    LOCAL CONST Robtarget Tr_meulage_motif_2_30 := [[-9.9900380859375,-86.177265625,6.42869384765625],[1.9380529697738E-05,0.00227567224534522,0.00851606674262758,-0.999961148018993],[0,0,0,0],[8.999999E+09,8.999999E+09,8.999999E+09,8.999999E+09,8.999999E+09,8.999999E+09]];
    LOCAL CONST Robtarget Tr_meulage_motif_2_31 := [[-10.2561494140625,-87.471703125,6.4017646484375],[1.9380529697738E-05,0.00227567224534522,0.00851606674262758,-0.999961148018993],[0,0,0,0],[8.999999E+09,8.999999E+09,8.999999E+09,8.999999E+09,8.999999E+09,8.999999E+09]];
    LOCAL CONST Robtarget Tr_meulage_motif_2_32 := [[-10.2795166015625,-88.7881796875,6.374595703125],[1.9380529697738E-05,0.00227567224534522,0.00851606674262758,-0.999961148018993],[0,0,0,0],[8.999999E+09,8.999999E+09,8.999999E+09,8.999999E+09,8.999999E+09,8.999999E+09]];
    LOCAL CONST Robtarget Tr_meulage_motif_2_33 := [[-10.16851953125,-89.573125,6.3585068359375],[1.9380529697738E-05,0.00227567224534522,0.00851606674262758,-0.999961148018993],[0,0,0,0],[8.999999E+09,8.999999E+09,8.999999E+09,8.999999E+09,8.999999E+09,8.999999E+09]];
    LOCAL CONST Robtarget Tr_meulage_motif_2_34 := [[-9.839921875,-90.785734375,6.333791015625],[1.9380529697738E-05,0.00227567224534522,0.00851606674262758,-0.999961148018993],[0,0,0,0],[8.999999E+09,8.999999E+09,8.999999E+09,8.999999E+09,8.999999E+09,8.999999E+09]];
    LOCAL CONST Robtarget Tr_meulage_motif_2_35 := [[-9.527951171875,-91.6141171875,6.316984375],[1.9380529697738E-05,0.00227567224534522,0.00851606674262758,-0.999961148018993],[0,0,0,0],[8.999999E+09,8.999999E+09,8.999999E+09,8.999999E+09,8.999999E+09,8.999999E+09]];
    LOCAL CONST Robtarget Tr_meulage_motif_2_36 := [[-9.115458984375,-92.4743359375,6.29960986328125],[1.9380529697738E-05,0.00227567224534522,0.00851606674262758,-0.999961148018993],[0,0,0,0],[8.999999E+09,8.999999E+09,8.999999E+09,8.999999E+09,8.999999E+09,8.999999E+09]];
    LOCAL CONST Robtarget Tr_meulage_motif_2_37 := [[-8.5968984375,-93.314609375,6.28274072265625],[1.9380529697738E-05,0.00227567224534522,0.00851606674262758,-0.999961148018993],[0,0,0,0],[8.999999E+09,8.999999E+09,8.999999E+09,8.999999E+09,8.999999E+09,8.999999E+09]];
    LOCAL CONST Robtarget Tr_meulage_motif_2_38 := [[-8.0731435546875,-94.1647890625,6.265671875],[1.9380529697738E-05,0.00227567224534522,0.00851606674262758,-0.999961148018993],[0,0,0,0],[8.999999E+09,8.999999E+09,8.999999E+09,8.999999E+09,8.999999E+09,8.999999E+09]];
    LOCAL CONST Robtarget Tr_meulage_motif_2_39 := [[-7.4576474609375,-94.9527734375,6.249966796875],[1.9380529697738E-05,0.00227567224534522,0.00851606674262758,-0.999961148018993],[0,0,0,0],[8.999999E+09,8.999999E+09,8.999999E+09,8.999999E+09,8.999999E+09,8.999999E+09]];
    LOCAL CONST Robtarget Tr_meulage_motif_2_40 := [[-6.84215185546875,-95.7407578125,6.23426220703125],[1.9380529697738E-05,0.00227567224534522,0.00851606674262758,-0.999961148018993],[0,0,0,0],[8.999999E+09,8.999999E+09,8.999999E+09,8.999999E+09,8.999999E+09,8.999999E+09]];
    LOCAL CONST Robtarget Tr_meulage_motif_2_41 := [[-6.22665576171875,-96.5287421875,6.21855712890625],[1.9380529697738E-05,0.00227567224534522,0.00851606674262758,-0.999961148018993],[0,0,0,0],[8.999999E+09,8.999999E+09,8.999999E+09,8.999999E+09,8.999999E+09,8.999999E+09]];
    LOCAL CONST Robtarget Tr_meulage_motif_2_42 := [[-5.61116015625,-97.3167265625,6.20285205078125],[1.9380529697738E-05,0.00227567224534522,0.00851606674262758,-0.999961148018993],[0,0,0,0],[8.999999E+09,8.999999E+09,8.999999E+09,8.999999E+09,8.999999E+09,8.999999E+09]];
    LOCAL CONST Robtarget Tr_meulage_motif_2_43 := [[-4.9956640625,-98.1047109375,6.18714697265625],[1.9380529697738E-05,0.00227567224534522,0.00851606674262758,-0.999961148018993],[0,0,0,0],[8.999999E+09,8.999999E+09,8.999999E+09,8.999999E+09,8.999999E+09,8.999999E+09]];
    LOCAL CONST Robtarget Tr_meulage_motif_2_44 := [[-4.38016796875,-98.8926953125,6.17144189453125],[1.9380529697738E-05,0.00227567224534522,0.00851606674262758,-0.999961148018993],[0,0,0,0],[8.999999E+09,8.999999E+09,8.999999E+09,8.999999E+09,8.999999E+09,8.999999E+09]];
    LOCAL CONST Robtarget Tr_meulage_motif_2_45 := [[-3.76467236328125,-99.680671875,6.15573681640625],[1.9380529697738E-05,0.00227567224534522,0.00851606674262758,-0.999961148018993],[0,0,0,0],[8.999999E+09,8.999999E+09,8.999999E+09,8.999999E+09,8.999999E+09,8.999999E+09]];
    LOCAL CONST Robtarget Tr_meulage_motif_2_46 := [[-3.14917651367188,-100.46865625,6.1400322265625],[1.9380529697738E-05,0.00227567224534522,0.00851606674262758,-0.999961148018993],[0,0,0,0],[8.999999E+09,8.999999E+09,8.999999E+09,8.999999E+09,8.999999E+09,8.999999E+09]];
    LOCAL CONST Robtarget Tr_meulage_motif_2_47 := [[-2.53368041992187,-101.256640625,6.1243271484375],[1.9380529697738E-05,0.00227567224534522,0.00851606674262758,-0.999961148018993],[0,0,0,0],[8.999999E+09,8.999999E+09,8.999999E+09,8.999999E+09,8.999999E+09,8.999999E+09]];
    LOCAL CONST Robtarget Tr_meulage_motif_2_48 := [[-1.91818469238281,-102.044625,6.1086220703125],[1.9380529697738E-05,0.00227567224534522,0.00851606674262758,-0.999961148018993],[0,0,0,0],[8.999999E+09,8.999999E+09,8.999999E+09,8.999999E+09,8.999999E+09,8.999999E+09]];
    LOCAL CONST Robtarget Tr_meulage_motif_2_49 := [[-1.39442980957031,-102.8948046875,6.09155322265625],[1.9380529697738E-05,0.00227567224534522,0.00851606674262758,-0.999961148018993],[0,0,0,0],[8.999999E+09,8.999999E+09,8.999999E+09,8.999999E+09,8.999999E+09,8.999999E+09]];
    LOCAL CONST Robtarget Tr_meulage_motif_2_50 := [[-0.978308227539063,-103.7705859375,6.073861328125],[1.9380529697738E-05,0.00227567224534522,0.00851606674262758,-0.999961148018993],[0,0,0,0],[8.999999E+09,8.999999E+09,8.999999E+09,8.999999E+09,8.999999E+09,8.999999E+09]];
    LOCAL CONST Robtarget Tr_meulage_motif_2_51 := [[-0.667714172363281,-104.6097890625,6.056830078125],[1.9380529697738E-05,0.00227567224534522,0.00851606674262758,-0.999961148018993],[0,0,0,0],[8.999999E+09,8.999999E+09,8.999999E+09,8.999999E+09,8.999999E+09,8.999999E+09]];
    LOCAL CONST Robtarget Tr_meulage_motif_2_52 := [[-0.469506439208984,-105.3576015625,6.041583984375],[1.9380529697738E-05,0.00227567224534522,0.00851606674262758,-0.999961148018993],[0,0,0,0],[8.999999E+09,8.999999E+09,8.999999E+09,8.999999E+09,8.999999E+09,8.999999E+09]];
    LOCAL CONST Robtarget Tr_meulage_motif_2_53 := [[-0.354962310791016,-106.5804375,6.01646826171875],[1.9380529697738E-05,0.00227567224534522,0.00851606674262758,-0.999961148018993],[0,0,0,0],[8.999999E+09,8.999999E+09,8.999999E+09,8.999999E+09,8.999999E+09,8.999999E+09]];
    LOCAL CONST Robtarget Tr_meulage_motif_2_54 := [[-0.510676147460937,-107.84615625,5.990228515625],[1.9380529697738E-05,0.00227567224534522,0.00851606674262758,-0.999961148018993],[0,0,0,0],[8.999999E+09,8.999999E+09,8.999999E+09,8.999999E+09,8.999999E+09,8.999999E+09]];
    LOCAL CONST Robtarget Tr_meulage_motif_2_55 := [[-1.00582373046875,-108.9113828125,5.9678232421875],[1.9380529697738E-05,0.00227567224534522,0.00851606674262758,-0.999961148018993],[0,0,0,0],[8.999999E+09,8.999999E+09,8.999999E+09,8.999999E+09,8.999999E+09,8.999999E+09]];
    LOCAL CONST Robtarget Tr_meulage_motif_2_56 := [[-1.43844482421875,-109.4835546875,5.95564111328125],[1.9380529697738E-05,0.00227567224534522,0.00851606674262758,-0.999961148018993],[0,0,0,0],[8.999999E+09,8.999999E+09,8.999999E+09,8.999999E+09,8.999999E+09,8.999999E+09]];
    LOCAL CONST Robtarget Tr_meulage_motif_2_57 := [[-2.00601672363281,-110.0076875,5.944330078125],[1.9380529697738E-05,0.00227567224534522,0.00851606674262758,-0.999961148018993],[0,0,0,0],[8.999999E+09,8.999999E+09,8.999999E+09,8.999999E+09,8.999999E+09,8.999999E+09]];
    LOCAL CONST Robtarget Tr_meulage_motif_2_58 := [[-2.6539853515625,-110.4286875,5.93507470703125],[1.9380529697738E-05,0.00227567224534522,0.00851606674262758,-0.999961148018993],[0,0,0,0],[8.999999E+09,8.999999E+09,8.999999E+09,8.999999E+09,8.999999E+09,8.999999E+09]];
    LOCAL CONST Robtarget Tr_meulage_motif_2_59 := [[-3.78569946289063,-110.780015625,5.92682763671875],[1.9380529697738E-05,0.00227567224534522,0.00851606674262758,-0.999961148018993],[0,0,0,0],[8.999999E+09,8.999999E+09,8.999999E+09,8.999999E+09,8.999999E+09,8.999999E+09]];
    LOCAL CONST Robtarget Tr_meulage_motif_2_60 := [[-4.502310546875,-110.8139453125,5.92549365234375],[1.9380529697738E-05,0.00227567224534522,0.00851606674262758,-0.999961148018993],[0,0,0,0],[8.999999E+09,8.999999E+09,8.999999E+09,8.999999E+09,8.999999E+09,8.999999E+09]];
    LOCAL CONST Robtarget Tr_meulage_motif_2_61 := [[-5.7475107421875,-110.660796875,5.9275498046875],[1.9380529697738E-05,0.00227567224534522,0.00851606674262758,-0.999961148018993],[0,0,0,0],[8.999999E+09,8.999999E+09,8.999999E+09,8.999999E+09,8.999999E+09,8.999999E+09]];
    LOCAL CONST Robtarget Tr_meulage_motif_2_62 := [[-6.43453515625,-110.454234375,5.93120166015625],[1.9380529697738E-05,0.00227567224534522,0.00851606674262758,-0.999961148018993],[0,0,0,0],[8.999999E+09,8.999999E+09,8.999999E+09,8.999999E+09,8.999999E+09,8.999999E+09]];
    LOCAL CONST Robtarget Tr_meulage_motif_2_63 := [[-7.55142333984375,-109.9081484375,5.94147412109375],[1.9380529697738E-05,0.00227567224534522,0.00851606674262758,-0.999961148018993],[0,0,0,0],[8.999999E+09,8.999999E+09,8.999999E+09,8.999999E+09,8.999999E+09,8.999999E+09]];
    LOCAL CONST Robtarget Tr_meulage_motif_2_64 := [[-8.29246875,-109.4394296875,5.950484375],[1.9380529697738E-05,0.00227567224534522,0.00851606674262758,-0.999961148018993],[0,0,0,0],[8.999999E+09,8.999999E+09,8.999999E+09,8.999999E+09,8.999999E+09,8.999999E+09]];
    LOCAL CONST Robtarget Tr_meulage_motif_2_65 := [[-9.0272607421875,-108.8308515625,5.9623837890625],[1.9380529697738E-05,0.00227567224534522,0.00851606674262758,-0.999961148018993],[0,0,0,0],[8.999999E+09,8.999999E+09,8.999999E+09,8.999999E+09,8.999999E+09,8.999999E+09]];
    LOCAL CONST Robtarget Tr_meulage_motif_2_66 := [[-9.7169951171875,-108.12421875,5.976345703125],[1.9380529697738E-05,0.00227567224534522,0.00851606674262758,-0.999961148018993],[0,0,0,0],[8.999999E+09,8.999999E+09,8.999999E+09,8.999999E+09,8.999999E+09,8.999999E+09]];
    LOCAL CONST Robtarget Tr_meulage_motif_2_67 := [[-10.415076171875,-107.4101484375,5.990453125],[1.9380529697738E-05,0.00227567224534522,0.00851606674262758,-0.999961148018993],[0,0,0,0],[8.999999E+09,8.999999E+09,8.999999E+09,8.999999E+09,8.999999E+09,8.999999E+09]];
    LOCAL CONST Robtarget Tr_meulage_motif_2_68 := [[-11.030572265625,-106.6221640625,6.006158203125],[1.9380529697738E-05,0.00227567224534522,0.00851606674262758,-0.999961148018993],[0,0,0,0],[8.999999E+09,8.999999E+09,8.999999E+09,8.999999E+09,8.999999E+09,8.999999E+09]];
    LOCAL CONST Robtarget Tr_meulage_motif_2_69 := [[-11.646068359375,-105.8341875,6.02186328125],[1.9380529697738E-05,0.00227567224534522,0.00851606674262758,-0.999961148018993],[0,0,0,0],[8.999999E+09,8.999999E+09,8.999999E+09,8.999999E+09,8.999999E+09,8.999999E+09]];
    LOCAL CONST Robtarget Tr_meulage_motif_2_70 := [[-12.261564453125,-105.046203125,6.037568359375],[1.9380529697738E-05,0.00227567224534522,0.00851606674262758,-0.999961148018993],[0,0,0,0],[8.999999E+09,8.999999E+09,8.999999E+09,8.999999E+09,8.999999E+09,8.999999E+09]];
    LOCAL CONST Robtarget Tr_meulage_motif_2_71 := [[-12.877060546875,-104.25821875,6.0532734375],[1.9380529697738E-05,0.00227567224534522,0.00851606674262758,-0.999961148018993],[0,0,0,0],[8.999999E+09,8.999999E+09,8.999999E+09,8.999999E+09,8.999999E+09,8.999999E+09]];
    LOCAL CONST Robtarget Tr_meulage_motif_2_72 := [[-13.4925556640625,-103.470234375,6.068978515625],[1.9380529697738E-05,0.00227567224534522,0.00851606674262758,-0.999961148018993],[0,0,0,0],[8.999999E+09,8.999999E+09,8.999999E+09,8.999999E+09,8.999999E+09,8.999999E+09]];
    LOCAL CONST Robtarget Tr_meulage_motif_2_73 := [[-14.1080517578125,-102.68225,6.08468359375],[1.9380529697738E-05,0.00227567224534522,0.00851606674262758,-0.999961148018993],[0,0,0,0],[8.999999E+09,8.999999E+09,8.999999E+09,8.999999E+09,8.999999E+09,8.999999E+09]];
    LOCAL CONST Robtarget Tr_meulage_motif_2_74 := [[-14.7235478515625,-101.894265625,6.10038818359375],[1.9380529697738E-05,0.00227567224534522,0.00851606674262758,-0.999961148018993],[0,0,0,0],[8.999999E+09,8.999999E+09,8.999999E+09,8.999999E+09,8.999999E+09,8.999999E+09]];
    LOCAL CONST Robtarget Tr_meulage_motif_2_75 := [[-15.3390439453125,-101.10628125,6.11609326171875],[1.9380529697738E-05,0.00227567224534522,0.00851606674262758,-0.999961148018993],[0,0,0,0],[8.999999E+09,8.999999E+09,8.999999E+09,8.999999E+09,8.999999E+09,8.999999E+09]];
    LOCAL CONST Robtarget Tr_meulage_motif_2_76 := [[-15.9545390625,-100.318296875,6.13179833984375],[1.9380529697738E-05,0.00227567224534522,0.00851606674262758,-0.999961148018993],[0,0,0,0],[8.999999E+09,8.999999E+09,8.999999E+09,8.999999E+09,8.999999E+09,8.999999E+09]];
    LOCAL CONST Robtarget Tr_meulage_motif_2_77 := [[-16.57003515625,-99.5303125,6.14750341796875],[1.9380529697738E-05,0.00227567224534522,0.00851606674262758,-0.999961148018993],[0,0,0,0],[8.999999E+09,8.999999E+09,8.999999E+09,8.999999E+09,8.999999E+09,8.999999E+09]];
    LOCAL CONST Robtarget Tr_meulage_motif_2_78 := [[-17.2681171875,-98.81625,6.16161083984375],[1.9380529697738E-05,0.00227567224534522,0.00851606674262758,-0.999961148018993],[0,0,0,0],[8.999999E+09,8.999999E+09,8.999999E+09,8.999999E+09,8.999999E+09,8.999999E+09]];
    LOCAL CONST Robtarget Tr_meulage_motif_2_79 := [[-18.01712890625,-98.200375,6.1736484375],[1.9380529697738E-05,0.00227567224534522,0.00851606674262758,-0.999961148018993],[0,0,0,0],[8.999999E+09,8.999999E+09,8.999999E+09,8.999999E+09,8.999999E+09,8.999999E+09]];
    LOCAL CONST Robtarget Tr_meulage_motif_2_80 := [[-18.756224609375,-97.6957265625,6.1834013671875],[1.9380529697738E-05,0.00227567224534522,0.00851606674262758,-0.999961148018993],[0,0,0,0],[8.999999E+09,8.999999E+09,8.999999E+09,8.999999E+09,8.999999E+09,8.999999E+09]];
    LOCAL CONST Robtarget Tr_meulage_motif_2_81 := [[-19.43528515625,-97.2745859375,6.19148486328125],[1.9380529697738E-05,0.00227567224534522,0.00851606674262758,-0.999961148018993],[0,0,0,0],[8.999999E+09,8.999999E+09,8.999999E+09,8.999999E+09,8.999999E+09,8.999999E+09]];
    LOCAL CONST Robtarget Tr_meulage_motif_2_82 := [[-20.598578125,-96.7861015625,6.20052880859375],[1.9380529697738E-05,0.00227567224534522,0.00851606674262758,-0.999961148018993],[0,0,0,0],[8.999999E+09,8.999999E+09,8.999999E+09,8.999999E+09,8.999999E+09,8.999999E+09]];
    LOCAL CONST Robtarget Tr_meulage_motif_2_83 := [[-21.892005859375,-96.582328125,6.20358642578125],[1.9380529697738E-05,0.00227567224534522,0.00851606674262758,-0.999961148018993],[0,0,0,0],[8.999999E+09,8.999999E+09,8.999999E+09,8.999999E+09,8.999999E+09,8.999999E+09]];
    LOCAL CONST Robtarget Tr_meulage_motif_2_84 := [[-23.12283984375,-96.7706171875,6.19861376953125],[1.9380529697738E-05,0.00227567224534522,0.00851606674262758,-0.999961148018993],[0,0,0,0],[8.999999E+09,8.999999E+09,8.999999E+09,8.999999E+09,8.999999E+09,8.999999E+09]];
    LOCAL CONST Robtarget Tr_meulage_motif_2_85 := [[-24.002875,-97.2429375,6.1880947265625],[1.9380529697738E-05,0.00227567224534522,0.00851606674262758,-0.999961148018993],[0,0,0,0],[8.999999E+09,8.999999E+09,8.999999E+09,8.999999E+09,8.999999E+09,8.999999E+09]];
    LOCAL CONST Robtarget Tr_meulage_motif_2_86 := [[-24.08325390625,-97.47246875,6.1832900390625],[1.9380529697738E-05,0.00227567224534522,0.00851606674262758,-0.999961148018993],[0,0,0,0],[8.999999E+09,8.999999E+09,8.999999E+09,8.999999E+09,8.999999E+09,8.999999E+09]];
    LOCAL CONST Robtarget Tr_meulage_motif_2_87 := [[-24.579828125,-98.0166796875,6.1716279296875],[1.9380529697738E-05,0.00227567224534522,0.00851606674262758,-0.999961148018993],[0,0,0,0],[8.999999E+09,8.999999E+09,8.999999E+09,8.999999E+09,8.999999E+09,8.999999E+09]];
    LOCAL CONST Robtarget Tr_meulage_motif_2_88 := [[-24.897240234375,-99.1321875,6.1483427734375],[1.9380529697738E-05,0.00227567224534522,0.00851606674262758,-0.999961148018993],[0,0,0,0],[8.999999E+09,8.999999E+09,8.999999E+09,8.999999E+09,8.999999E+09,8.999999E+09]];
    LOCAL CONST Robtarget Tr_meulage_motif_2_89 := [[-24.91957421875,-99.8569921875,6.13337646484375],[1.9380529697738E-05,0.00227567224534522,0.00851606674262758,-0.999961148018993],[0,0,0,0],[8.999999E+09,8.999999E+09,8.999999E+09,8.999999E+09,8.999999E+09,8.999999E+09]];
    LOCAL CONST Robtarget Tr_meulage_motif_2_90 := [[-24.6419296875,-101.0740625,6.1085234375],[1.9380529697738E-05,0.00227567224534522,0.00851606674262758,-0.999961148018993],[0,0,0,0],[8.999999E+09,8.999999E+09,8.999999E+09,8.999999E+09,8.999999E+09,8.999999E+09]];
    LOCAL CONST Robtarget Tr_meulage_motif_2_91 := [[-24.329958984375,-101.9024453125,6.091716796875],[1.9380529697738E-05,0.00227567224534522,0.00851606674262758,-0.999961148018993],[0,0,0,0],[8.999999E+09,8.999999E+09,8.999999E+09,8.999999E+09,8.999999E+09,8.999999E+09]];
    LOCAL CONST Robtarget Tr_meulage_motif_2_92 := [[-23.917466796875,-102.7626640625,6.07434228515625],[1.9380529697738E-05,0.00227567224534522,0.00851606674262758,-0.999961148018993],[0,0,0,0],[8.999999E+09,8.999999E+09,8.999999E+09,8.999999E+09,8.999999E+09,8.999999E+09]];
    LOCAL CONST Robtarget Tr_meulage_motif_2_93 := [[-23.39890625,-103.6029453125,6.05747314453125],[1.9380529697738E-05,0.00227567224534522,0.00851606674262758,-0.999961148018993],[0,0,0,0],[8.999999E+09,8.999999E+09,8.999999E+09,8.999999E+09,8.999999E+09,8.999999E+09]];
    LOCAL CONST Robtarget Tr_meulage_motif_2_94 := [[-22.87515234375,-104.453125,6.040404296875],[1.9380529697738E-05,0.00227567224534522,0.00851606674262758,-0.999961148018993],[0,0,0,0],[8.999999E+09,8.999999E+09,8.999999E+09,8.999999E+09,8.999999E+09,8.999999E+09]];
    LOCAL CONST Robtarget Tr_meulage_motif_2_95 := [[-22.25965625,-105.241109375,6.02469921875],[1.9380529697738E-05,0.00227567224534522,0.00851606674262758,-0.999961148018993],[0,0,0,0],[8.999999E+09,8.999999E+09,8.999999E+09,8.999999E+09,8.999999E+09,8.999999E+09]];
    LOCAL CONST Robtarget Tr_meulage_motif_2_96 := [[-21.64416015625,-106.0290859375,6.00899462890625],[1.9380529697738E-05,0.00227567224534522,0.00851606674262758,-0.999961148018993],[0,0,0,0],[8.999999E+09,8.999999E+09,8.999999E+09,8.999999E+09,8.999999E+09,8.999999E+09]];
    LOCAL CONST Robtarget Tr_meulage_motif_2_97 := [[-21.0286640625,-106.8170703125,5.99328955078125],[1.9380529697738E-05,0.00227567224534522,0.00851606674262758,-0.999961148018993],[0,0,0,0],[8.999999E+09,8.999999E+09,8.999999E+09,8.999999E+09,8.999999E+09,8.999999E+09]];
    LOCAL CONST Robtarget Tr_meulage_motif_2_98 := [[-20.41316796875,-107.6050546875,5.97758447265625],[1.9380529697738E-05,0.00227567224534522,0.00851606674262758,-0.999961148018993],[0,0,0,0],[8.999999E+09,8.999999E+09,8.999999E+09,8.999999E+09,8.999999E+09,8.999999E+09]];
    LOCAL CONST Robtarget Tr_meulage_motif_2_99 := [[-19.797671875,-108.3930390625,5.96187939453125],[1.9380529697738E-05,0.00227567224534522,0.00851606674262758,-0.999961148018993],[0,0,0,0],[8.999999E+09,8.999999E+09,8.999999E+09,8.999999E+09,8.999999E+09,8.999999E+09]];
    LOCAL CONST Robtarget Tr_meulage_motif_2_100 := [[-19.182177734375,-109.1810234375,5.94617431640625],[1.9380529697738E-05,0.00227567224534522,0.00851606674262758,-0.999961148018993],[0,0,0,0],[8.999999E+09,8.999999E+09,8.999999E+09,8.999999E+09,8.999999E+09,8.999999E+09]];
    LOCAL CONST Robtarget Tr_meulage_motif_2_101 := [[-18.566681640625,-109.9690078125,5.93046923828125],[1.9380529697738E-05,0.00227567224534522,0.00851606674262758,-0.999961148018993],[0,0,0,0],[8.999999E+09,8.999999E+09,8.999999E+09,8.999999E+09,8.999999E+09,8.999999E+09]];
    LOCAL CONST Robtarget Tr_meulage_motif_2_102 := [[-17.951185546875,-110.7569921875,5.9147646484375],[1.9380529697738E-05,0.00227567224534522,0.00851606674262758,-0.999961148018993],[0,0,0,0],[8.999999E+09,8.999999E+09,8.999999E+09,8.999999E+09,8.999999E+09,8.999999E+09]];
    LOCAL CONST Robtarget Tr_meulage_motif_2_103 := [[-17.335689453125,-111.5449765625,5.8990595703125],[1.9380529697738E-05,0.00227567224534522,0.00851606674262758,-0.999961148018993],[0,0,0,0],[8.999999E+09,8.999999E+09,8.999999E+09,8.999999E+09,8.999999E+09,8.999999E+09]];
    LOCAL CONST Robtarget Tr_meulage_motif_2_104 := [[-16.720193359375,-112.3329609375,5.8833544921875],[1.9380529697738E-05,0.00227567224534522,0.00851606674262758,-0.999961148018993],[0,0,0,0],[8.999999E+09,8.999999E+09,8.999999E+09,8.999999E+09,8.999999E+09,8.999999E+09]];
    LOCAL CONST Robtarget Tr_meulage_motif_2_105 := [[-16.104697265625,-113.1209453125,5.8676494140625],[1.9380529697738E-05,0.00227567224534522,0.00851606674262758,-0.999961148018993],[0,0,0,0],[8.999999E+09,8.999999E+09,8.999999E+09,8.999999E+09,8.999999E+09,8.999999E+09]];
    LOCAL CONST Robtarget Tr_meulage_motif_2_106 := [[-15.4892021484375,-113.9089296875,5.8519443359375],[1.9380529697738E-05,0.00227567224534522,0.00851606674262758,-0.999961148018993],[0,0,0,0],[8.999999E+09,8.999999E+09,8.999999E+09,8.999999E+09,8.999999E+09,8.999999E+09]];
    LOCAL CONST Robtarget Tr_meulage_motif_2_107 := [[-14.8737060546875,-114.69690625,5.8362392578125],[1.9380529697738E-05,0.00227567224534522,0.00851606674262758,-0.999961148018993],[0,0,0,0],[8.999999E+09,8.999999E+09,8.999999E+09,8.999999E+09,8.999999E+09,8.999999E+09]];
    LOCAL CONST Robtarget Tr_meulage_motif_2_108 := [[-14.2582099609375,-115.484890625,5.8205341796875],[1.9380529697738E-05,0.00227567224534522,0.00851606674262758,-0.999961148018993],[0,0,0,0],[8.999999E+09,8.999999E+09,8.999999E+09,8.999999E+09,8.999999E+09,8.999999E+09]];
    LOCAL CONST Robtarget Tr_meulage_motif_2_109 := [[-13.6427138671875,-116.272875,5.80482958984375],[1.9380529697738E-05,0.00227567224534522,0.00851606674262758,-0.999961148018993],[0,0,0,0],[8.999999E+09,8.999999E+09,8.999999E+09,8.999999E+09,8.999999E+09,8.999999E+09]];
    LOCAL CONST Robtarget Tr_meulage_motif_2_110 := [[-13.0272177734375,-117.060859375,5.78912451171875],[1.9380529697738E-05,0.00227567224534522,0.00851606674262758,-0.999961148018993],[0,0,0,0],[8.999999E+09,8.999999E+09,8.999999E+09,8.999999E+09,8.999999E+09,8.999999E+09]];
    LOCAL CONST Robtarget Tr_meulage_motif_2_111 := [[-12.41172265625,-117.84884375,5.77341943359375],[1.9380529697738E-05,0.00227567224534522,0.00851606674262758,-0.999961148018993],[0,0,0,0],[8.999999E+09,8.999999E+09,8.999999E+09,8.999999E+09,8.999999E+09,8.999999E+09]];
    LOCAL CONST Robtarget Tr_meulage_motif_2_112 := [[-11.7962265625,-118.636828125,5.75771435546875],[1.9380529697738E-05,0.00227567224534522,0.00851606674262758,-0.999961148018993],[0,0,0,0],[8.999999E+09,8.999999E+09,8.999999E+09,8.999999E+09,8.999999E+09,8.999999E+09]];
    LOCAL CONST Robtarget Tr_meulage_motif_2_113 := [[-11.18073046875,-119.4248125,5.74200927734375],[1.9380529697738E-05,0.00227567224534522,0.00851606674262758,-0.999961148018993],[0,0,0,0],[8.999999E+09,8.999999E+09,8.999999E+09,8.999999E+09,8.999999E+09,8.999999E+09]];
    LOCAL CONST Robtarget Tr_meulage_motif_2_114 := [[-10.565234375,-120.212796875,5.72630419921875],[1.9380529697738E-05,0.00227567224534522,0.00851606674262758,-0.999961148018993],[0,0,0,0],[8.999999E+09,8.999999E+09,8.999999E+09,8.999999E+09,8.999999E+09,8.999999E+09]];
    LOCAL CONST Robtarget Tr_meulage_motif_2_115 := [[-9.94973828125,-121.00078125,5.71059912109375],[1.9380529697738E-05,0.00227567224534522,0.00851606674262758,-0.999961148018993],[0,0,0,0],[8.999999E+09,8.999999E+09,8.999999E+09,8.999999E+09,8.999999E+09,8.999999E+09]];

